TYPE ST_S7_Incoming_Cyclic :
STRUCT
	by1 AT%I* 	: BYTE;
	b1 AT%I* 	: BOOL;
	b2 AT%I* 	: BOOL;
	b3 AT%I* 	: BOOL;
	b4 AT%I* 	: BOOL;
	w1 AT%I*	: DWORD;
	r1 AT%I*	: REAL;
	r2 AT%I*	: REAL;
	i1 AT%I*	: INT;	
END_STRUCT
END_TYPE

(* stored: Version 1.1.0.1, ProductVersion 3.1.4024.11
   DUT ST_S7_Incoming_Cyclic: Id {1e14f928-5fde-4d18-aec1-2af0d8ea36ef} *)
